Staubli VAL3: modelParmIdent.pgx

public program modelParmIdent(ModelParameter& x_mImpedParm)
  local num l_n
begin

  //This program is used for identifying the robot impedance model parameters or other model parameters on line
  //in realtime. And the identified model parameters are used for robot realtime control based on the relevant
  //models. For now, the impedance model parameters are identified in this program.

  //Impedance model parameter identification
  //Suppose the static parameter for impedance model in six dimensions.
  //Mass Parameter(Unit: N*s^2/m, N*s^2/°)
  for l_n=0 to 2
    x_mImpedParm.MassParm[l_n]=0.1
    x_mImpedParm.MassParm[l_n+3]=0.00005
  endFor
  //Damping Parameter(Unit: N*s/m, N*s/°)
  for l_n=0 to 2
    x_mImpedParm.DampingParm[l_n]=4
    x_mImpedParm.DampingParm[l_n+3]=4
  endFor
  //Stiffness Parameter(Unit: N/m, N/°)
  for l_n=0 to 2
    x_mImpedParm.StiffnessParm[l_n]=4
    x_mImpedParm.StiffnessParm[l_n+3]=4
  endFor

  //Other model parameter identification

end
